Fanuc KAREL source: compact_preamble.KL

PROGRAM IO0201
%NOLOCKGROUP
ROUTINE RTEST
VAR
L1 : ARRAY[3] OF INTEGER;L2 : XYZWPR
L3 : JOINTPOS9
L4 : POSITION
S1:INTEGER
S2:INTEGER
A:REAL
B:BOOLEAN
C:REAL
BEGIN
S1=1
L1[1]=2
B=TRUE
C=1.0
SET_POS_REG(S1,L2,S2,1)
END RTEST
BEGIN
RTEST
END IO0201
